(* PLC project Programme MGS_2-07_refactorJOY.project, CODESYS CODESYS V3.5 SP19 Patch 1 *)
(* stored: creationDateTime 2026-06-29T23:37:38.7086223, modificationDateTime 2026-06-29T22:49:33.424 *)

PROGRAM PLC_PRG_MAIN
  VAR
    InstanceSafety : FB_Safety;
    InstanceJoystick : FB_Joystick;
    LocalEmergencyStopTOR : BOOL := TRUE;
  END_VAR

            // PROGRAM PLC_PRG

// 1. ÉVALUATION DE LA SÉCURITÉ TRANSVERSE
InstanceSafety(
    Enable := TRUE,
    EStopArmed := LocalEmergencyStopTOR,
    CanOnline := diagCAN.IsOnline,
    CanOperational := diagCAN.IsOperational,
    EthercatOk := LocalEthercatOk
);

// 2. ACQUISITION DU GESTE OPÉRATEUR SÉCURISÉ
InstanceJoystick(
    Enable := TRUE,
    SafeStop := InstanceSafety.SafeStop,   // Reçoit la sécurité positive inversée
    SafetyOk := InstanceSafety.SafetyOk,   // Reçoit le feu vert global
    CanOnline := diagCAN.IsOnline,
    CanOperational := diagCAN.IsOperational,
    RawX := JoyXRaw_ANA1,
    RawY := JoyYRaw_ANA2,
    RawButton := JoyBtnRaw
);
          
END_PROGRAM
